// Setpoints for the lasers
TYPE ST_LaserSetpoints :
STRUCT
    {attribute 'pytmc' := '
        pv: MIN_VOLTAGE
        io: io
        field: EGU Volts
    '}
    nMinVoltage : LREAL; // Minimum voltage the laser will be allowed to operate at
    {attribute 'pytmc' := '
        pv: MIN_NOMINAL_VOLTAGE
        io: io
        field: EGU Volts
    '}
    nMinNominalVoltage : LREAL; // Minimum voltage for the laser to be operating nominally
END_STRUCT
END_TYPE

(* stored: Version 1.1.0.1, ProductVersion 3.1.4022.18
   DUT ST_LaserSetpoints: Id {2d3526ec-8638-4f89-a072-c7f0a369da3b} *)
